% RSLogix 500 project Project_5.RSS, saved by version 8.30.00.16 %
PROJECT "UNTITLED"    % processor: Bul.1763 MicroLogix 1100 Series B %

PROGRAM FILES
  LAD 2   7 rungs

DATA FILES
  O0 OUTPUT  4 elements
  I1 INPUT  6 elements
  S2 STATUS  66 elements
  B3 BINARY  1 elements
  T4 TIMER  2 elements
  C5 COUNTER  1 elements
  R6 CONTROL  1 elements
  N7 INTEGER  1 elements
  F8 FLOAT  1 elements

LADDER 2
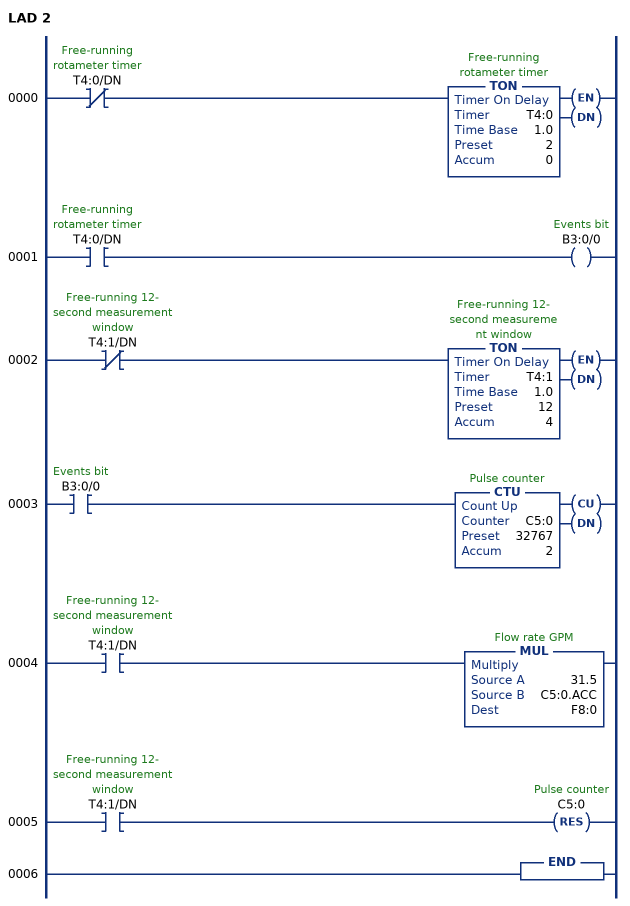
% Rung: 0 %
SOR XIO T4:0/DN TON T4:0 1.0 2 0 EOR
%   T4:0  "Free-running rotameter timer" %
% Rung: 1 %
SOR XIC T4:0/DN OTE B3:0/0 EOR
%   T4:0  "Free-running rotameter timer" %
%   B3:0/0  "Events bit" %
% Rung: 2 %
SOR XIO T4:1/DN TON T4:1 1.0 12 4 EOR
%   T4:1  "Free-running 12- second measurement window" %
% Rung: 3 %
SOR XIC B3:0/0 CTU C5:0 32767 2 EOR
%   B3:0/0  "Events bit" %
%   C5:0  "Pulse counter" %
% Rung: 4 %
SOR XIC T4:1/DN MUL 31.5 C5:0.ACC F8:0 EOR
%   T4:1  "Free-running 12- second measurement window" %
%   C5:0.ACC  "Pulse counter" %
%   F8:0  "Flow rate GPM" %
% Rung: 5 %
SOR XIC T4:1/DN RES C5:0 EOR
%   T4:1  "Free-running 12- second measurement window" %
%   C5:0  "Pulse counter" %
% Rung: 6 %
SOR END EOR

DATA TABLE (non-zero values as saved)
DATA T4
% .PRE .ACC %
% T4:0 % 2 0
% T4:1 % 12 5
DATA C5
% .PRE .ACC %
% C5:0 % 32767 2
DATA F8
% F8:0 % 189
